FUNCTION_BLOCK FB_CTUD_ULINT (* Up Down counter *)
  (* Standard: 61499-1; Description: Copyright (c) 2023 Martin Erich Jobst This program and the accompanying materials are made available under the terms of the Eclipse Public License 2.0 which is available at https://www.eclipse.org/legal/epl-2.0/ SPDX-License-Identifier: EPL-2.0 *)
  (* Version 1.0, 2023-04-28, Martin Jobst *)
  (* Version 3.0, 2025-04-14, Patrick Aigner, changed package *)
  PACKAGE iec61131::counters;
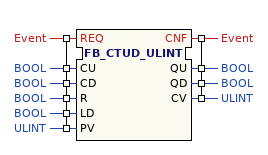
  EVENT_INPUT
    REQ WITH CU, CD, R, LD, PV; (* Normal Execution Request *)
  END_EVENT
  EVENT_OUTPUT
    CNF WITH QU, QD, CV; (* Execution Confirmation *)
  END_EVENT
  VAR_INPUT
    CU : BOOL; (* Count up *)
    CD : BOOL; (* Count down *)
    R : BOOL; (* Reset *)
    LD : BOOL; (* Load *)
    PV : ULINT; (* Preset value *)
  END_VAR
  VAR_OUTPUT
    QU : BOOL; (* Output up *)
    QD : BOOL; (* Output down *)
    CV : ULINT; (* Count value *)
  END_VAR
  ALGORITHM REQ IN ST:
IF R THEN
  CV := 0;
ELSE
  IF LD THEN
    CV := PV;
  ELSE
    IF NOT(CU AND CD) THEN
      IF CU AND CV < 18446744073709551615 THEN
        CV := CV + 1;
      ELSIF CD AND CV > 0 THEN
        CV := CV - 1;
      END_IF;
    END_IF;
  END_IF;
END_IF;
QU := CV >= PV;
QD := CV <= 0;
  END_ALGORITHM
END_FUNCTION_BLOCK
